(* IEC 61131-3 sources: RL_MAR/experiments/comparison/llm4plc/results/gpt-4o_20260507_114630/20260507_114857, 1 file *)

(* ---- generated_code_iteration_0.st ---- *)
START_ST
FUNCTION_BLOCK FB_BatchAnalogConverter
VAR_INPUT
    count : INT; // Number of channels to process (maximum 10)
    analogValues : ARRAY[1..10] OF REAL; // Array of analog input values
END_VAR

VAR_OUTPUT
    channel_enable : ARRAY[1..10] OF BOOL; // Enable conversion for each channel
    channel_hiLIM : ARRAY[1..10] OF REAL; // Upper limit for scaling
    channel_loLIM : ARRAY[1..10] OF REAL; // Lower limit for scaling
    channel_bipolar : ARRAY[1..10] OF BOOL; // TRUE for bipolar, FALSE for unipolar
    channel_measuringMode : ARRAY[1..10] OF INT; // Measurement mode (0, 1, or 2)
    channel_retVal : ARRAY[1..10] OF WORD; // Status information for each channel
    channel_outputValue : ARRAY[1..10] OF REAL; // Converted output values
END_VAR

VAR
    i : INT; // Loop index for iterating through channels
    scaledValue : REAL; // Temporary variable for holding scaled values during processing
END_VAR

// Iterate through each channel
FOR i := 1 TO count DO
    // Initialize default return value
    channel_retVal[i] := 0;

    // Check if the channel is enabled
    IF channel_enable[i] THEN
        // Check for valid measuring mode
        CASE channel_measuringMode[i] OF
            0: // Non-temperature measurement
                // Check if the channel is unipolar or bipolar
                IF channel_bipolar[i] THEN
                    // Bipolar: Map analogValues from -27648.0 to 27648.0 to channel_loLIM to channel_hiLIM
                    scaledValue := ((analogValues[i] + 27648.0) / 55296.0) * (channel_hiLIM[i] - channel_loLIM[i]) + channel_loLIM[i];
                ELSE
                    // Unipolar: Map analogValues from 0.0 to 27648.0 to channel_loLIM to channel_hiLIM
                    scaledValue := (analogValues[i] / 27648.0) * (channel_hiLIM[i] - channel_loLIM[i]) + channel_loLIM[i];
                END_IF;
                channel_outputValue[i] := scaledValue;
            1: // Standard temperature measurement
                // Set output value to one-tenth of analogValues
                channel_outputValue[i] := analogValues[i] / 10.0;
            2: // Climatic temperature measurement
                // Set output value to one-hundredth of analogValues
                channel_outputValue[i] := analogValues[i] / 100.0;
            ELSE
                // Invalid measuring mode
                channel_retVal[i] := 16#8001; // Error code for invalid mode
        END_CASE;

        // Error check: Validate scaling limits
        IF channel_hiLIM[i] <= channel_loLIM[i] THEN
            channel_retVal[i] := 16#8002; // Error code for invalid limits
        END_IF;
    END_IF;
END_FOR;
END_FUNCTION_BLOCK
END_ST
